PROGRAM MAIN
VAR
	COUNTER : UDINT ;
END_VAR

IF GVL.S1 AND GVL.S2 THEN
	GVL.LED1 := TRUE;
	GVL.LED2 := FALSE;
	//COUNTER := COUNTER +1 ;
ELSIF NOT( GVL.S1 AND GVL.S2) THEN
	GVL.LED1 := FALSE;
	GVL.LED2 := TRUE;
	
	
END_IF

GVL.counter := GVL.counter +1 ;

IF GVL.counter > 10000 THEN
	GVL.counter := 0;
	
END_IF

END_PROGRAM

(* stored: Version 1.1.0.1, ProductVersion 3.1.4024.12
   POU MAIN: Id {22e85fc1-0839-443f-ba5e-12789aeaecdd}, SpecialFunc None *)
